// Mitsubishi GX Works2 project: TEx02   PLC: Q02/Q02H

PROGRAM MAIN
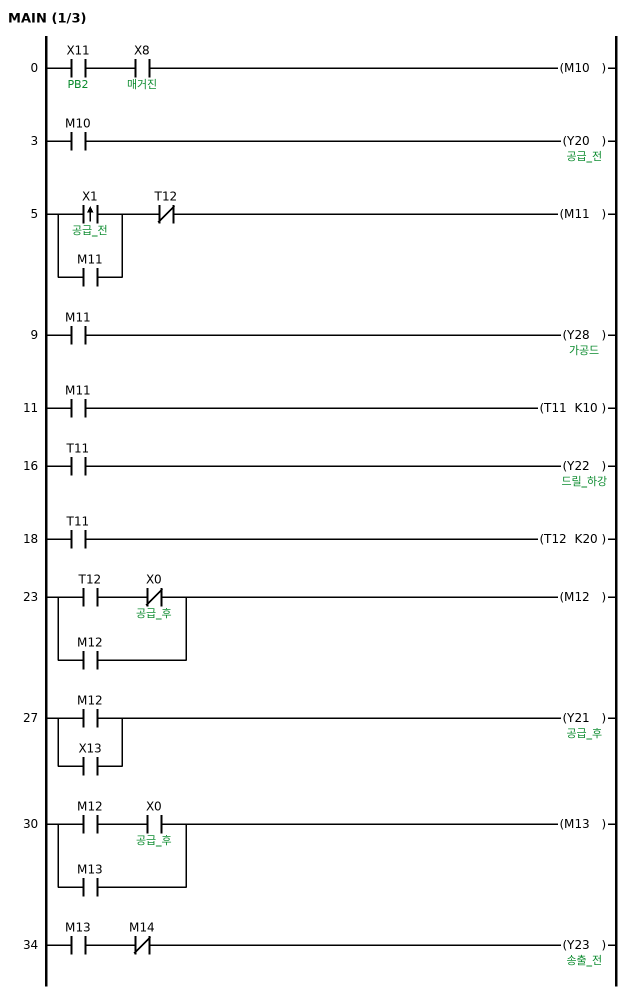
0     LD      X11  ; PB2
      AND     X8  ; 매거진
      OUT     M10
3     LD      M10
      OUT     Y20  ; 공급_전
5     LDP     X1  ; 공급_전
      OR      M11
      ANI     T12
      OUT     M11
9     LD      M11
      OUT     Y28  ; 가공드
11    LD      M11
      OUT     T11 K10
16    LD      T11
      OUT     Y22  ; 드릴_하강
18    LD      T11
      OUT     T12 K20
23    LD      T12
      ANI     X0  ; 공급_후
      OR      M12
      OUT     M12
27    LD      M12
      OR      X13
      OUT     Y21  ; 공급_후
30    LD      M12
      AND     X0  ; 공급_후
      OR      M13
      OUT     M13
34    LD      M13
      ANI     M14
      OUT     Y23  ; 송출_전
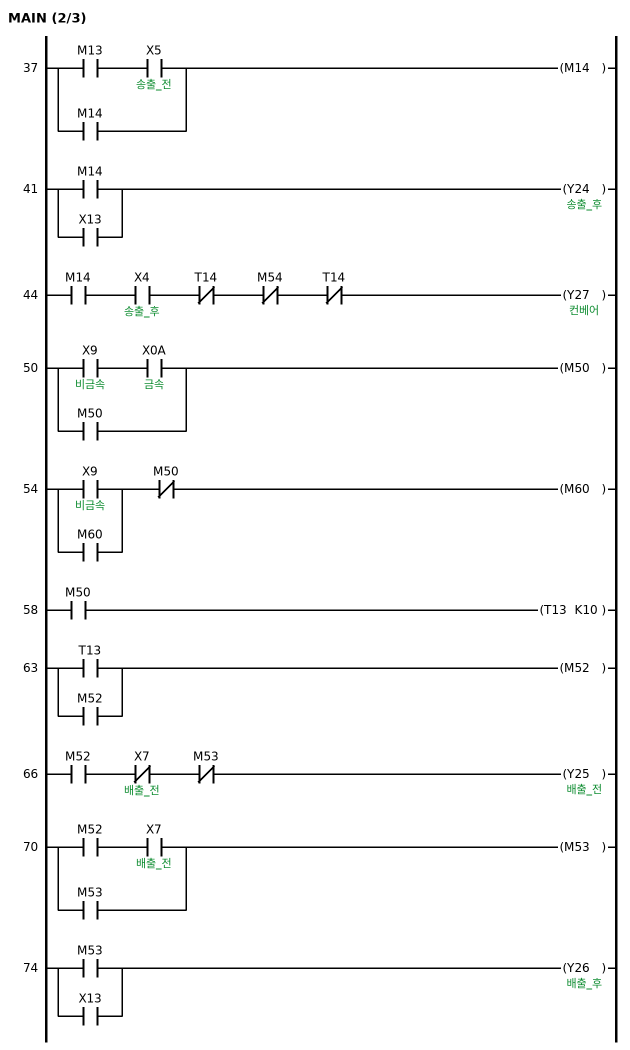
37    LD      M13
      AND     X5  ; 송출_전
      OR      M14
      OUT     M14
41    LD      M14
      OR      X13
      OUT     Y24  ; 송출_후
44    LD      M14
      AND     X4  ; 송출_후
      ANI     T14
      ANI     M54
      ANI     T14
      OUT     Y27  ; 컨베어
50    LD      X9  ; 비금속
      AND     X0A  ; 금속
      OR      M50
      OUT     M50
54    LD      X9  ; 비금속
      OR      M60
      ANI     M50
      OUT     M60
58    LD      M50
      OUT     T13 K10
63    LD      T13
      OR      M52
      OUT     M52
66    LD      M52
      ANI     X7  ; 배출_전
      ANI     M53
      OUT     Y25  ; 배출_전
70    LD      M52
      AND     X7  ; 배출_전
      OR      M53
      OUT     M53
74    LD      M53
      OR      X13
      OUT     Y26  ; 배출_후
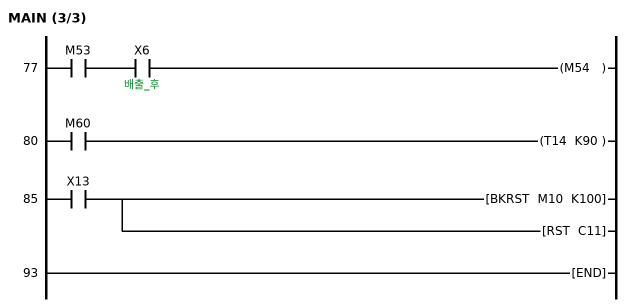
77    LD      M53
      AND     X6  ; 배출_후
      OUT     M54
80    LD      M60
      OUT     T14 K90
85    LD      X13
      BKRST   M10 K100
      RST     C11
93    END
END_PROGRAM

// device comments not shown above
X2  ; 드릴_상
X3  ; 드릴_하
X10  ; PB1
X12  ; PB3
Y29  ; 적색
Y2A  ; 황색
Y2B  ; 녹색
